(*
SPDX-FileCopyrightText: © 2026 Oleksandr Tiutyk <trofimich@gmail.com>
SPDX-License-Identifier: MIT
License: https://opensource.org/license/mit
*)

INTERFACE IEmptyException EXTENDS IException

END_INTERFACE

(* stored: Version 1.1.0.1
   Itf IEmptyException: Id {17176714-5c64-47e1-941b-1bed8926f011} *)
